// EL5101 | 1-channel incremental encoder terminal, 5V, RS422
FUNCTION_BLOCK EL5101

VAR_INPUT
	En				: BOOL;
	iTerminal_ID	: INT;
	ErrorSystem		: POINTER TO ST_ErrorSystem;
END_VAR

VAR_OUTPUT
	EnO		: BOOL;
	bError	: BOOL;
END_VAR

VAR
	//WC_State is handled by NC, so NOT included here.
	InfoData_State		AT %I* : UINT;
	
	//FB-s
	EL5101_Error	: FB_TerminalError;
END_VAR

(*
* TODO: Channel Status word (Connected to NC -> Not needed )
*)
EnO:=En;

//Error FB instances
EL5101_Error(
	En					:= TRUE,
	iTerminal_ID		:= iTerminal_ID,
	bWcState			:= FALSE,
	uiInfoData_State	:= InfoData_State,
	pErrorSystem		:= ErrorSystem,
	bError 				=> bError,
);

END_FUNCTION_BLOCK

(* stored: Version 1.1.0.1, ProductVersion 3.1.4022.18
   POU EL5101: Id {5df30a0c-1331-4fa2-acfe-28b08cfc5f04}, SpecialFunc None *)
